Fanuc KAREL source: wusetimeshft.kl

PROGRAM wusetimeshft
%NOLOCKGROUP
VAR
  p : POSITION
  q : POSITION
  i : INTEGER
  r : REAL
BEGIN
  WITH $USETIMESHFT = TRUE MOVE TO p
END wusetimeshft
